FUNCTION_BLOCK EcMasterFrameCount IMPLEMENTS IEcTask
VAR_INPUT
END_VAR
VAR_OUTPUT
END_VAR
VAR
	iState : INT;
	masterFrameCount : Tc2_EtherCAT.FB_EcMasterFrameCount;
	_execute: BOOL;
	_done: BOOL;
	_busy: BOOL;
	_error: BOOL;
	_netId: AMSNETID;
END_VAR

CASE iState OF
	0:
		IF _execute THEN
			_done := FALSE;
			_busy := TRUE;
			_error := FALSE;
			masterFrameCount.bExecute := TRUE;
			IF masterFrameCount.bBusy THEN
				iState := 10;
				_execute := false;
			END_IF
		END_IF
	10:
		IF NOT masterFrameCount.bBusy THEN
			IF NOT masterFrameCount.bError THEN
				_done := TRUE;
			ELSE
				_error := TRUE;
			END_IF
			_busy := FALSE;
			masterFrameCount.bExecute := FALSE;
			iState := 0;
		END_IF
END_CASE

masterFrameCount(sNetId := Tc2_System.F_CreateAmsNetId(nIds := NetId));

{warning 'add method implementation '}
METHOD Abort : BOOL
masterFrameCount.bExecute := FALSE;
_busy := FALSE;
_execute := FALSE;
Abort := TRUE;
iState := 0;
END_METHOD

{warning 'add property implementation'}
PROPERTY Busy : BOOL
GET
Busy := _busy;
END_GET
END_PROPERTY

{warning 'add property implementation'}
PROPERTY Done : BOOL
GET
Done := _done;
END_GET
END_PROPERTY

{warning 'add property implementation'}
PROPERTY Error : BOOL
GET
Error := _error;
END_GET
END_PROPERTY

{warning 'add method implementation '}
METHOD Execute : BOOL
IF NOT masterFrameCount.bBusy THEN
	Execute := _execute := True;
END_IF
END_METHOD

PROPERTY FrameNumber : UDINT
GET
FrameNumber := masterFrameCount.nFrames;
END_GET
END_PROPERTY

{warning 'add property implementation'}
PROPERTY NetID : amsnetid
GET
NetID := _netId;
END_GET
SET
_netId := NetID;
END_SET
END_PROPERTY

END_FUNCTION_BLOCK

(* stored: Version 1.1.0.1, ProductVersion 3.1.4024.9
   POU EcMasterFrameCount: Id {58af2663-b399-4f8e-9118-545ee07dec25}, SpecialFunc None
   Method Abort: Id {79fe29ad-a018-4ec2-a476-8187f5ed3f81}
   Property Busy: Id {ae21d882-3963-4a99-a796-2f6660c32adf}
   Get Get: Id {7b539d48-054b-40f2-9b10-ed8a64b76468}
   Property Done: Id {c89ecd70-5537-4a02-a79b-408824e02475}
   Get Get: Id {a27c6fb5-f0c9-47fb-8691-13bc23b66e6a}
   Property Error: Id {934fcbec-b834-43ff-85f0-a0dba8d81326}
   Get Get: Id {6c2de2b0-3d83-4cd6-8054-b2873daf398f}
   Method Execute: Id {b305b830-562e-4f96-8de5-06a5cbe6af19}
   Property FrameNumber: Id {3814b406-1e13-4d18-891b-ef3d014103c2}
   Get Get: Id {f663a3ad-ba87-4e25-a345-8364b87a69d5}
   Property NetID: Id {01a37ee7-2252-4d39-bcdd-53cdc7b6da81}
   Get Get: Id {d82e447b-cd62-4a5a-bfe3-c5f066cd5e45}
   Set Set: Id {77ece9b7-b565-4d3c-9c92-ad87e585ddd2} *)
